(* IEC 61131-3 sources: STruCpp-cpp/stdfb, 4 files *)

(* ---- bistable.st ---- *)
(* IEC 61131-3 Standard Function Blocks: Bistable Latches *)

FUNCTION_BLOCK SR
  VAR_INPUT S1, R : BOOL; END_VAR
  VAR_OUTPUT Q1 : BOOL; END_VAR
  Q1 := S1 OR ((NOT R) AND Q1);
END_FUNCTION_BLOCK

FUNCTION_BLOCK RS
  VAR_INPUT S, R1 : BOOL; END_VAR
  VAR_OUTPUT Q1 : BOOL; END_VAR
  Q1 := (NOT R1) AND (S OR Q1);
END_FUNCTION_BLOCK

(* ---- counter.st ---- *)
(* IEC 61131-3 Standard Function Blocks: Counters *)

FUNCTION_BLOCK CTU
  VAR_INPUT
    CU : BOOL;
    R : BOOL;
    PV : INT;
  END_VAR
  VAR_OUTPUT
    Q : BOOL;
    CV : INT;
  END_VAR
  VAR
    CU_T : R_TRIG;
  END_VAR
  CU_T(CLK := CU);
  IF R THEN
    CV := 0;
  ELSIF CU_T.Q AND (CV < PV) THEN
    CV := CV + 1;
  END_IF;
  Q := (CV >= PV);
END_FUNCTION_BLOCK

FUNCTION_BLOCK CTD
  VAR_INPUT
    CD : BOOL;
    LD : BOOL;
    PV : INT;
  END_VAR
  VAR_OUTPUT
    Q : BOOL;
    CV : INT;
  END_VAR
  VAR
    CD_T : F_TRIG;
  END_VAR
  CD_T(CLK := CD);
  IF LD THEN
    CV := PV;
  ELSIF CD_T.Q AND (CV > 0) THEN
    CV := CV - 1;
  END_IF;
  Q := (CV <= 0);
END_FUNCTION_BLOCK

FUNCTION_BLOCK CTUD
  VAR_INPUT
    CU : BOOL;
    CD : BOOL;
    R : BOOL;
    LD : BOOL;
    PV : INT;
  END_VAR
  VAR_OUTPUT
    QU : BOOL;
    QD : BOOL;
    CV : INT;
  END_VAR
  VAR
    CU_T : R_TRIG;
    CD_T : F_TRIG;
  END_VAR
  CU_T(CLK := CU);
  CD_T(CLK := CD);
  IF R THEN
    CV := 0;
  ELSIF LD THEN
    CV := PV;
  ELSE
    IF CU_T.Q AND (CV < PV) THEN
      CV := CV + 1;
    END_IF;
    IF CD_T.Q AND (CV > 0) THEN
      CV := CV - 1;
    END_IF;
  END_IF;
  QU := (CV >= PV);
  QD := (CV <= 0);
END_FUNCTION_BLOCK

FUNCTION_BLOCK CTU_DINT
  VAR_INPUT
    CU : BOOL;
    R : BOOL;
    PV : DINT;
  END_VAR
  VAR_OUTPUT
    Q : BOOL;
    CV : DINT;
  END_VAR
  VAR
    CU_T : R_TRIG;
  END_VAR
  CU_T(CLK := CU);
  IF R THEN
    CV := 0;
  ELSIF CU_T.Q AND (CV < PV) THEN
    CV := CV + 1;
  END_IF;
  Q := (CV >= PV);
END_FUNCTION_BLOCK

FUNCTION_BLOCK CTU_LINT
  VAR_INPUT
    CU : BOOL;
    R : BOOL;
    PV : LINT;
  END_VAR
  VAR_OUTPUT
    Q : BOOL;
    CV : LINT;
  END_VAR
  VAR
    CU_T : R_TRIG;
  END_VAR
  CU_T(CLK := CU);
  IF R THEN
    CV := 0;
  ELSIF CU_T.Q AND (CV < PV) THEN
    CV := CV + 1;
  END_IF;
  Q := (CV >= PV);
END_FUNCTION_BLOCK

FUNCTION_BLOCK CTU_UDINT
  VAR_INPUT
    CU : BOOL;
    R : BOOL;
    PV : UDINT;
  END_VAR
  VAR_OUTPUT
    Q : BOOL;
    CV : UDINT;
  END_VAR
  VAR
    CU_T : R_TRIG;
  END_VAR
  CU_T(CLK := CU);
  IF R THEN
    CV := 0;
  ELSIF CU_T.Q AND (CV < PV) THEN
    CV := CV + 1;
  END_IF;
  Q := (CV >= PV);
END_FUNCTION_BLOCK

FUNCTION_BLOCK CTU_ULINT
  VAR_INPUT
    CU : BOOL;
    R : BOOL;
    PV : ULINT;
  END_VAR
  VAR_OUTPUT
    Q : BOOL;
    CV : ULINT;
  END_VAR
  VAR
    CU_T : R_TRIG;
  END_VAR
  CU_T(CLK := CU);
  IF R THEN
    CV := 0;
  ELSIF CU_T.Q AND (CV < PV) THEN
    CV := CV + 1;
  END_IF;
  Q := (CV >= PV);
END_FUNCTION_BLOCK

FUNCTION_BLOCK CTD_DINT
  VAR_INPUT
    CD : BOOL;
    LD : BOOL;
    PV : DINT;
  END_VAR
  VAR_OUTPUT
    Q : BOOL;
    CV : DINT;
  END_VAR
  VAR
    CD_T : F_TRIG;
  END_VAR
  CD_T(CLK := CD);
  IF LD THEN
    CV := PV;
  ELSIF CD_T.Q AND (CV > 0) THEN
    CV := CV - 1;
  END_IF;
  Q := (CV <= 0);
END_FUNCTION_BLOCK

FUNCTION_BLOCK CTD_LINT
  VAR_INPUT
    CD : BOOL;
    LD : BOOL;
    PV : LINT;
  END_VAR
  VAR_OUTPUT
    Q : BOOL;
    CV : LINT;
  END_VAR
  VAR
    CD_T : F_TRIG;
  END_VAR
  CD_T(CLK := CD);
  IF LD THEN
    CV := PV;
  ELSIF CD_T.Q AND (CV > 0) THEN
    CV := CV - 1;
  END_IF;
  Q := (CV <= 0);
END_FUNCTION_BLOCK

FUNCTION_BLOCK CTD_UDINT
  VAR_INPUT
    CD : BOOL;
    LD : BOOL;
    PV : UDINT;
  END_VAR
  VAR_OUTPUT
    Q : BOOL;
    CV : UDINT;
  END_VAR
  VAR
    CD_T : F_TRIG;
  END_VAR
  CD_T(CLK := CD);
  IF LD THEN
    CV := PV;
  ELSIF CD_T.Q AND (CV > 0) THEN
    CV := CV - 1;
  END_IF;
  Q := (CV <= 0);
END_FUNCTION_BLOCK

FUNCTION_BLOCK CTD_ULINT
  VAR_INPUT
    CD : BOOL;
    LD : BOOL;
    PV : ULINT;
  END_VAR
  VAR_OUTPUT
    Q : BOOL;
    CV : ULINT;
  END_VAR
  VAR
    CD_T : F_TRIG;
  END_VAR
  CD_T(CLK := CD);
  IF LD THEN
    CV := PV;
  ELSIF CD_T.Q AND (CV > 0) THEN
    CV := CV - 1;
  END_IF;
  Q := (CV <= 0);
END_FUNCTION_BLOCK

FUNCTION_BLOCK CTUD_DINT
  VAR_INPUT
    CU : BOOL;
    CD : BOOL;
    R : BOOL;
    LD : BOOL;
    PV : DINT;
  END_VAR
  VAR_OUTPUT
    QU : BOOL;
    QD : BOOL;
    CV : DINT;
  END_VAR
  VAR
    CU_T : R_TRIG;
    CD_T : F_TRIG;
  END_VAR
  CU_T(CLK := CU);
  CD_T(CLK := CD);
  IF R THEN
    CV := 0;
  ELSIF LD THEN
    CV := PV;
  ELSE
    IF CU_T.Q AND (CV < PV) THEN
      CV := CV + 1;
    END_IF;
    IF CD_T.Q AND (CV > 0) THEN
      CV := CV - 1;
    END_IF;
  END_IF;
  QU := (CV >= PV);
  QD := (CV <= 0);
END_FUNCTION_BLOCK

FUNCTION_BLOCK CTUD_LINT
  VAR_INPUT
    CU : BOOL;
    CD : BOOL;
    R : BOOL;
    LD : BOOL;
    PV : LINT;
  END_VAR
  VAR_OUTPUT
    QU : BOOL;
    QD : BOOL;
    CV : LINT;
  END_VAR
  VAR
    CU_T : R_TRIG;
    CD_T : F_TRIG;
  END_VAR
  CU_T(CLK := CU);
  CD_T(CLK := CD);
  IF R THEN
    CV := 0;
  ELSIF LD THEN
    CV := PV;
  ELSE
    IF CU_T.Q AND (CV < PV) THEN
      CV := CV + 1;
    END_IF;
    IF CD_T.Q AND (CV > 0) THEN
      CV := CV - 1;
    END_IF;
  END_IF;
  QU := (CV >= PV);
  QD := (CV <= 0);
END_FUNCTION_BLOCK

FUNCTION_BLOCK CTUD_UDINT
  VAR_INPUT
    CU : BOOL;
    CD : BOOL;
    R : BOOL;
    LD : BOOL;
    PV : UDINT;
  END_VAR
  VAR_OUTPUT
    QU : BOOL;
    QD : BOOL;
    CV : UDINT;
  END_VAR
  VAR
    CU_T : R_TRIG;
    CD_T : F_TRIG;
  END_VAR
  CU_T(CLK := CU);
  CD_T(CLK := CD);
  IF R THEN
    CV := 0;
  ELSIF LD THEN
    CV := PV;
  ELSE
    IF CU_T.Q AND (CV < PV) THEN
      CV := CV + 1;
    END_IF;
    IF CD_T.Q AND (CV > 0) THEN
      CV := CV - 1;
    END_IF;
  END_IF;
  QU := (CV >= PV);
  QD := (CV <= 0);
END_FUNCTION_BLOCK

FUNCTION_BLOCK CTUD_ULINT
  VAR_INPUT
    CU : BOOL;
    CD : BOOL;
    R : BOOL;
    LD : BOOL;
    PV : ULINT;
  END_VAR
  VAR_OUTPUT
    QU : BOOL;
    QD : BOOL;
    CV : ULINT;
  END_VAR
  VAR
    CU_T : R_TRIG;
    CD_T : F_TRIG;
  END_VAR
  CU_T(CLK := CU);
  CD_T(CLK := CD);
  IF R THEN
    CV := 0;
  ELSIF LD THEN
    CV := PV;
  ELSE
    IF CU_T.Q AND (CV < PV) THEN
      CV := CV + 1;
    END_IF;
    IF CD_T.Q AND (CV > 0) THEN
      CV := CV - 1;
    END_IF;
  END_IF;
  QU := (CV >= PV);
  QD := (CV <= 0);
END_FUNCTION_BLOCK

(* ---- edge_detection.st ---- *)
(* IEC 61131-3 Standard Function Blocks: Edge Detection *)

FUNCTION_BLOCK R_TRIG
  VAR_INPUT CLK : BOOL; END_VAR
  VAR_OUTPUT Q : BOOL; END_VAR
  VAR RETAIN M : BOOL; END_VAR
  Q := CLK AND NOT M;
  M := CLK;
END_FUNCTION_BLOCK

FUNCTION_BLOCK F_TRIG
  VAR_INPUT CLK : BOOL; END_VAR
  VAR_OUTPUT Q : BOOL; END_VAR
  VAR RETAIN M : BOOL := TRUE; END_VAR
  Q := NOT CLK AND NOT M;
  M := NOT CLK;
END_FUNCTION_BLOCK

(* ---- timer.st ---- *)
(* IEC 61131-3 Standard Function Blocks: Timers *)
(* Uses TIME() built-in function for current time (CODESYS-compatible) *)

FUNCTION_BLOCK TON
  VAR_INPUT
    IN : BOOL;
    PT : TIME;
  END_VAR
  VAR_OUTPUT
    Q : BOOL;
    ET : TIME;
  END_VAR
  VAR
    STATE : SINT;
    PREV_IN : BOOL;
    CURRENT_TIME, START_TIME : TIME;
  END_VAR

  CURRENT_TIME := TIME();

  IF ((STATE = 0) AND NOT(PREV_IN) AND IN) THEN
    STATE := 1;
    Q := FALSE;
    START_TIME := CURRENT_TIME;
  ELSE
    IF (NOT(IN)) THEN
      ET := T#0s;
      Q := FALSE;
      STATE := 0;
    ELSIF (STATE = 1) THEN
      IF ((START_TIME + PT) <= CURRENT_TIME) THEN
        STATE := 2;
        Q := TRUE;
        ET := PT;
      ELSE
        ET := CURRENT_TIME - START_TIME;
      END_IF;
    END_IF;
  END_IF;

  PREV_IN := IN;
END_FUNCTION_BLOCK

FUNCTION_BLOCK TOF
  VAR_INPUT
    IN : BOOL;
    PT : TIME;
  END_VAR
  VAR_OUTPUT
    Q : BOOL;
    ET : TIME;
  END_VAR
  VAR
    STATE : SINT;
    PREV_IN : BOOL;
    CURRENT_TIME, START_TIME : TIME;
  END_VAR

  CURRENT_TIME := TIME();

  IF ((STATE = 0) AND PREV_IN AND NOT(IN)) THEN
    STATE := 1;
    START_TIME := CURRENT_TIME;
  ELSE
    IF (IN) THEN
      ET := T#0s;
      Q := TRUE;
      STATE := 0;
    ELSIF (STATE = 1) THEN
      IF ((START_TIME + PT) <= CURRENT_TIME) THEN
        STATE := 2;
        Q := FALSE;
        ET := PT;
      ELSE
        Q := TRUE;
        ET := CURRENT_TIME - START_TIME;
      END_IF;
    END_IF;
  END_IF;

  PREV_IN := IN;
END_FUNCTION_BLOCK

FUNCTION_BLOCK TP
  VAR_INPUT
    IN : BOOL;
    PT : TIME;
  END_VAR
  VAR_OUTPUT
    Q : BOOL;
    ET : TIME;
  END_VAR
  VAR
    STATE : SINT;
    PREV_IN : BOOL;
    CURRENT_TIME, START_TIME : TIME;
  END_VAR

  CURRENT_TIME := TIME();

  IF ((STATE = 0) AND NOT(PREV_IN) AND IN) THEN
    STATE := 1;
    Q := TRUE;
    START_TIME := CURRENT_TIME;
  ELSIF (STATE = 1) THEN
    IF ((START_TIME + PT) <= CURRENT_TIME) THEN
      STATE := 2;
      Q := FALSE;
      ET := PT;
    ELSE
      ET := CURRENT_TIME - START_TIME;
    END_IF;
  END_IF;

  IF (NOT(IN) AND (STATE = 2)) THEN
    STATE := 0;
    ET := T#0s;
  END_IF;

  PREV_IN := IN;
END_FUNCTION_BLOCK
